(* CODESYS project GVL_STATISTIC.gvl.xml

Project tree, tasks and I/O mapping:
  global variables GVL_STATISTIC
*)

// GVL_STATISTIC
{attribute 'qualified_only'}
VAR_GLOBAL
	stStatistic			: ST_STATISTIC;
END_VAR
